{attribute 'GeneratedUsingTerminal: EP1312-0001-0016'}
{attribute addProperty BoxType "EP1312-0001-0016"}
{attribute addProperty Id "InfoDataAT %I*InfoData_6F19DB2B2"}
{attribute addProperty CRC "532711307"}
{attribute addProperty Size "2"}
TYPE EP1312_1FC0878B EXTENDS EtcSlaveTerminalBase_947E5A46 :
STRUCT
	{attribute addProperty Name "InfoData"}
	InfoData : InfoData_6F19DB2B;
END_STRUCT
END_TYPE

(* stored: Version 1.2.0.0, ProductVersion 3.1.4024.9
   DUT EP1312_1FC0878B: Id {78b62b8c-b984-440d-abf2-08d4ebb1a0b7} *)
